FUNCTION_BLOCK CU00xSuspendTask EXTENDS CUBaseSuspend IMPLEMENTS ICUTask
VAR

	
	
	_sb : TcoCore.StringBuilder;
END_VAR

VAR

END_VAR

Run();

(*~
	<docu>
		<summary>
			Main method of the sequener. Custom code needs to be placed here. The sequencer is executed by call of **Instance.Run()** method.
			This method is abstract, and it must be overridden in derived block.
		</summary>
	</docu>
~*)
METHOD PROTECTED Main : BOOL
(*

	SUSPEND PROCESS 
	Following steps provide suspend actions for this controlled unit.
	Add components add write customized sequence according to your need.
*)

		
//
IF (Step(100, TRUE, '<#WAITING FOR START#>')) THEN
    //-------------------------------------    

    StepCompleteWhen(TRUE);
    //-------------------------------------
END_IF

//HERE  YOU CAN WRITE  WHAT IS NECESSARY 
//TO SUPSEND  PROCESS..... TO INTERUPT SAFETY

IF (Step(1000, TRUE, '<#SUSPENDING COMPONENTS#>')) THEN
 	//-------------------------------------    
	//StepCompleteWhen(Station.AutomatTask.CurrentStep.Status <> eStepStatus.Running);
		
  	StepCompleteWhen(CurrentStep.Duration >= T#3000MS);
    //-------------------------------------
END_IF

IF (Step(30000, TRUE, 'SUSPEND DONE')) THEN
    //-------------------------------------
		
        THIS^._done:=TRUE;
		THIS^.Task.DoneWhen(TRUE);
		
   
    //-------------------------------------	
END_IF
END_METHOD

METHOD PUBLIC OnStart
SUPER^.OnStart();
Station.RecoverTask.Restore();
END_METHOD

PROPERTY Station : REFERENCE TO CU00x
GET
VAR
    _station : POINTER TO CU00x;
END_VAR
IF __QUERYPOINTER(Parent, _station) THEN // Check if _Parent is Station001
    Station REF= _station^;              // If the check is successful dereference a pointer. simlar to THIS^ or SUPER^
END_IF
END_GET
END_PROPERTY

END_FUNCTION_BLOCK

(* stored: Version 1.1.0.1
   POU CU00xSuspendTask: Id {6dd32787-25bd-4e8d-99a8-0cfb2f9159ea}, SpecialFunc None
   Method Main: Id {b0a4a57f-1d5a-4900-afa9-341f96856d5c}
   Method OnStart: Id {f9ce7e5a-b25e-4c30-bea4-590e14b7f0c4}
   Property Station: Id {2e84916a-2a86-4cff-a2a2-8f0af095939f}
   Get Get: Id {1b0f1dbd-05b6-4e4d-ba90-424ceaba6669} *)
